VAR_GLOBAL
	OffloadStart:BOOL;
END_VAR

(* stored: Version 1.1.0.1, ProductVersion 3.1.0.36
   GVL GVL_Offload: Id {7c24a32e-32c9-45cc-ad89-55ee864705ee} *)
